FUNCTION F_ToAnyBit : T_AnyBit
VAR_INPUT
    anyBit	: ANY_BIT;
END_VAR

F_ToAnyBit := anyBit;

END_FUNCTION

(* stored: Version 1.1.0.1
   POU F_ToAnyBit: Id {c8c93c83-3030-4fbf-9a70-9cab4e4d19a9}, SpecialFunc None *)
